FUNCTION TryConvert_UDINT_TO_USINT : BOOL
VAR_INPUT
	in : UDINT;
	out : REFERENCE TO USINT;
END_VAR

IF in > DatatypeLimits.MAX_VALUE_OF_UDINT_WHICH_CAN_BE_HELD_IN_A_USINT THEN
	RETURN;
END_IF

out := UDINT_TO_USINT(in);
TryConvert_UDINT_TO_USINT := TRUE;

END_FUNCTION

(* stored: Version 1.1.0.1, ProductVersion 3.1.4024.12
   POU TryConvert_UDINT_TO_USINT: Id {d16686bd-78f6-475d-8b77-5a40c0cae6b5}, SpecialFunc None *)
